FUNCTION_BLOCK InfoDataAdsDC EXTENDS InfoDataAds
VAR
	_dcOutputShift AT %I* :   DINT;
	_dcInputShift AT %I* :   DINT;
END_VAR

PROPERTY DcInputShift : DINT
GET
DcInputShift := _dcInputShift;
END_GET
END_PROPERTY

PROPERTY DcOutputShift : DINT
GET
DcOutputShift := _dcOutputShift;
END_GET
END_PROPERTY

END_FUNCTION_BLOCK

(* stored: Version 1.1.0.1, ProductVersion 3.1.4024.9
   POU InfoDataAdsDC: Id {85d853e3-99bf-0cd8-3bfe-085d8909bd22}, SpecialFunc None
   Property DcInputShift: Id {f5a572ff-2fdd-0c7f-02f8-33b0a027cec4}
   Get Get: Id {263460f9-927d-0426-1f0e-021570ad314b}
   Property DcOutputShift: Id {53c4d525-cf73-0ad5-0251-a661daa8c505}
   Get Get: Id {30465fde-abac-0c23-3d7d-554ad3ee5414} *)
